FUNCTION_BLOCK ContactorNO
VAR
	output AT %Q* : BOOL;
END_VAR

METHOD Close
VAR_INPUT
END_VAR
output := TRUE;
END_METHOD

PROPERTY IsClose : BOOL
GET
IsClose := output;
END_GET
END_PROPERTY

PROPERTY IsOpen : BOOL
GET
IsOpen := NOT output;
END_GET
END_PROPERTY

METHOD Open
VAR_INPUT
END_VAR
output := FALSE;
END_METHOD

END_FUNCTION_BLOCK

(* stored: Version 1.1.0.1, ProductVersion 3.1.4024.12
   POU ContactorNO: Id {34f17846-6c9c-439c-a272-47f598c34ff1}, SpecialFunc None
   Method Close: Id {5c1b5935-8b86-4af1-9876-0d6cb3a73a8c}
   Property IsClose: Id {9777f89f-26f2-411d-9e89-f23cb119cd23}
   Get Get: Id {93db381f-214a-4f2d-aede-1ececcdbf29a}
   Property IsOpen: Id {1387b2a5-bb72-4e4e-bbb4-3c813c4c5dc2}
   Get Get: Id {f428f270-3002-477c-bb31-f7a57cc71eaa}
   Method Open: Id {6f58826d-db61-431a-8618-806e742a33b9} *)
